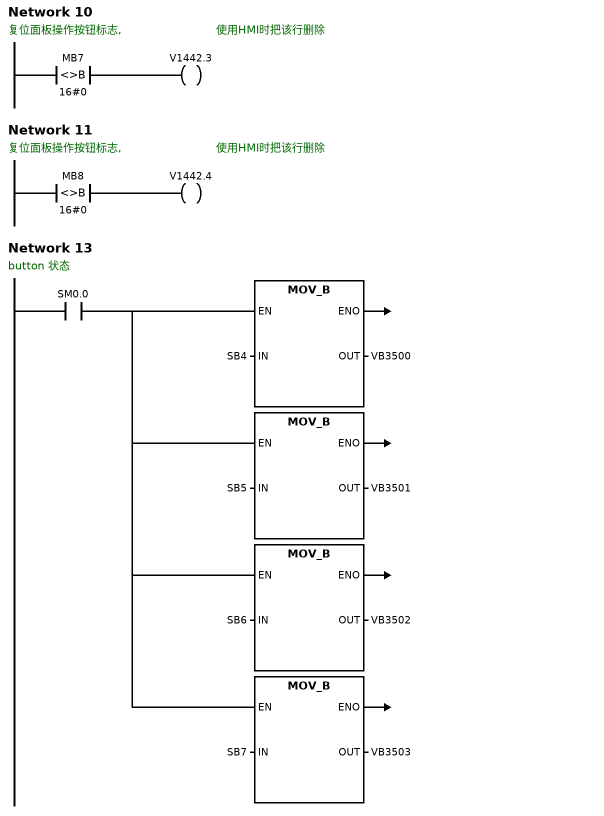
[picture p72: SBR17 networks 10-13]
Network 10
// 复位面板操作按钮标志,                           使用HMI时把该行删除
LDB<>  MB7, 16#0
=      V1442.3
Network 11
// 复位面板操作按钮标志,                           使用HMI时把该行删除
LDB<>  MB8, 16#0
=      V1442.4
Network 13
// button 状态
LD     SM0.0
MOVB   SB4, VB3500
MOVB   SB5, VB3501
MOVB   SB6, VB3502
MOVB   SB7, VB3503
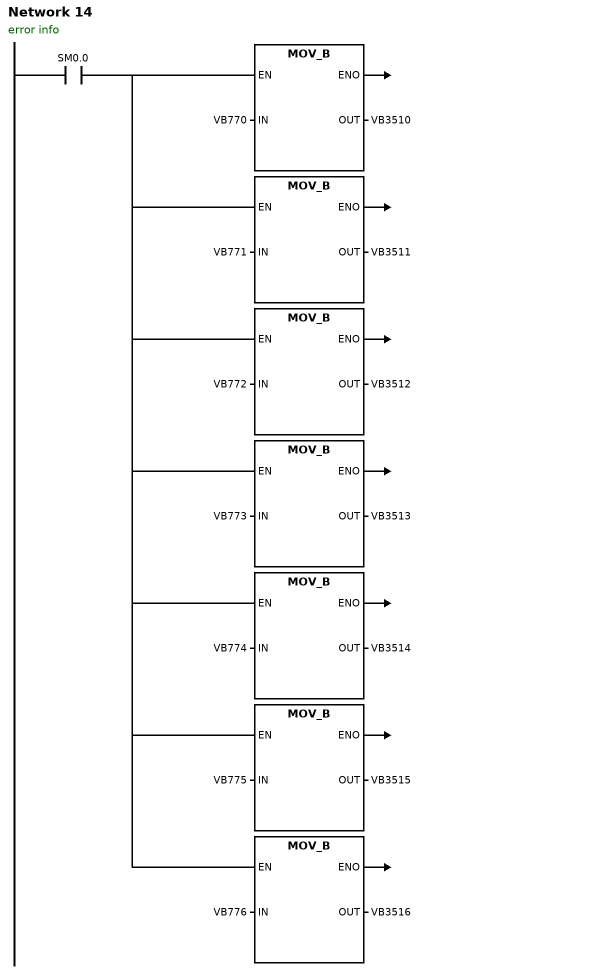
Network 14
// error info
LD     SM0.0
MOVB   VB770, VB3510
MOVB   VB771, VB3511
MOVB   VB772, VB3512
MOVB   VB773, VB3513
MOVB   VB774, VB3514
MOVB   VB775, VB3515
MOVB   VB776, VB3516
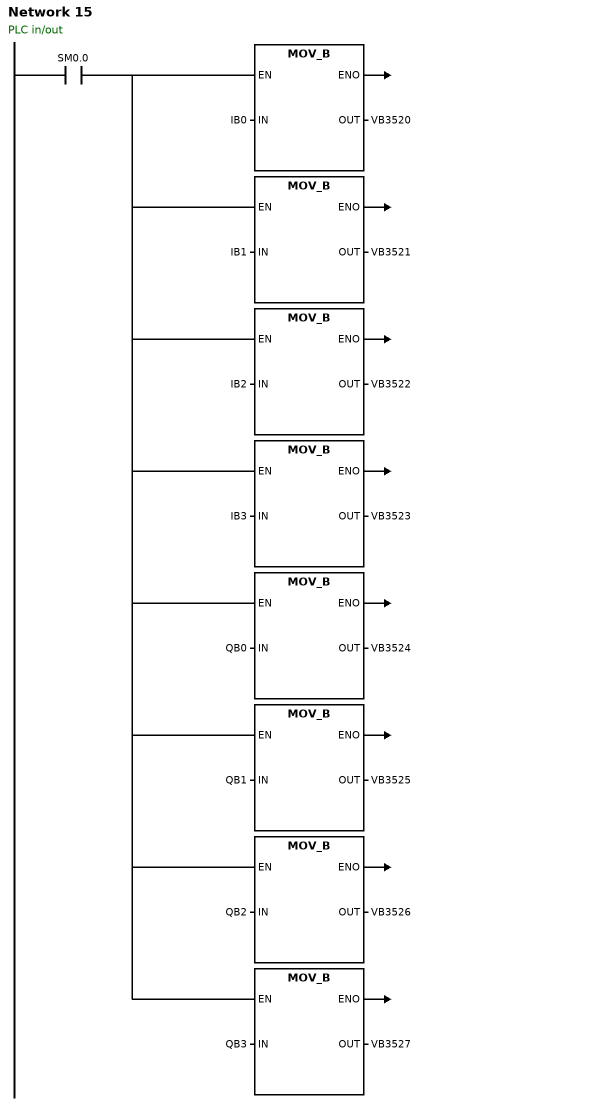
Network 15
// PLC in/out
LD     SM0.0
MOVB   IB0, VB3520
MOVB   IB1, VB3521
MOVB   IB2, VB3522
MOVB   IB3, VB3523
MOVB   QB0, VB3524
MOVB   QB1, VB3525
MOVB   QB2, VB3526
MOVB   QB3, VB3527
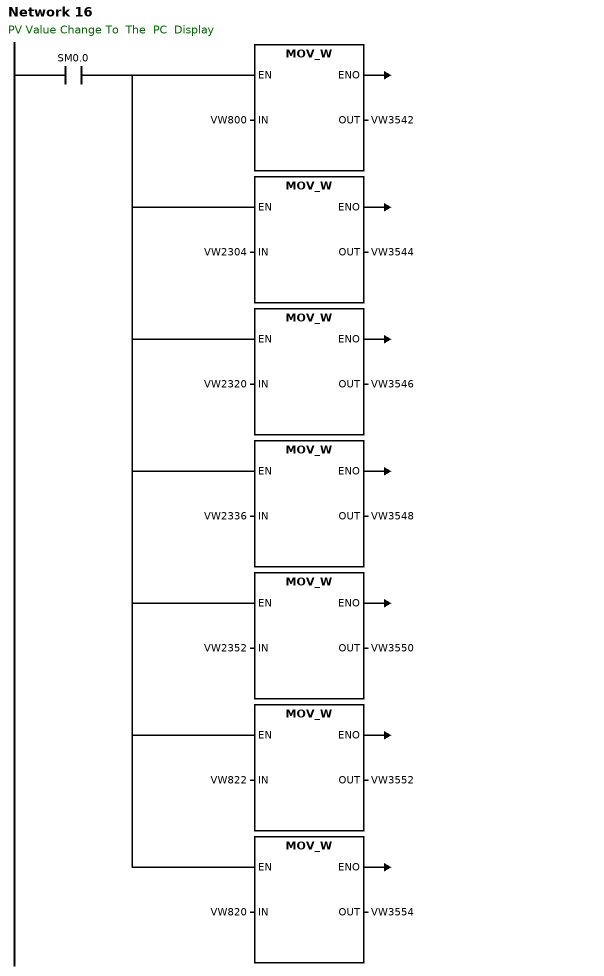
Network 16
// PV Value Change To  The  PC  Display 
LD     SM0.0
MOVW   VW800, VW3542
MOVW   VW2304, VW3544
MOVW   VW2320, VW3546
MOVW   VW2336, VW3548
MOVW   VW2352, VW3550
MOVW   VW822, VW3552
MOVW   VW820, VW3554
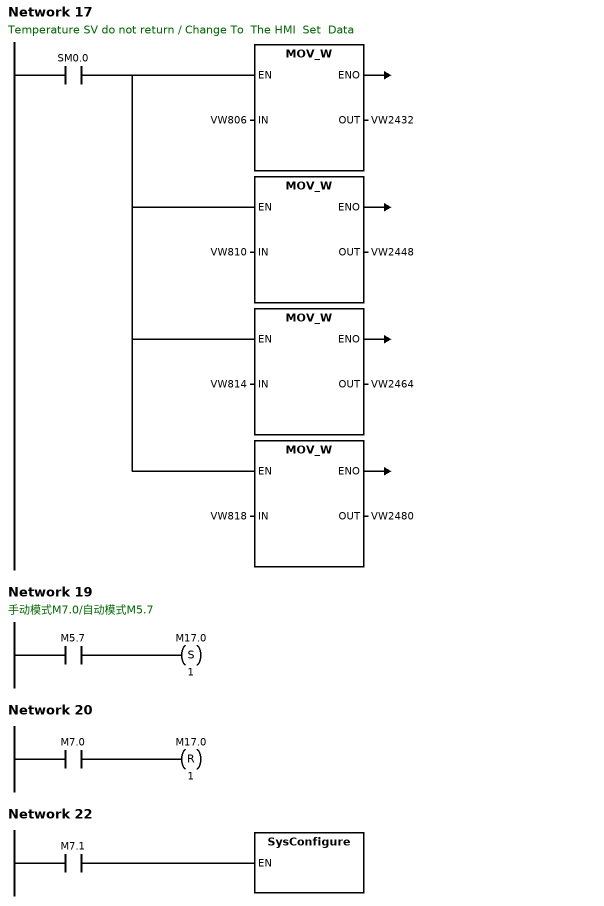
Network 17
// Temperature SV do not return
// Change To  The HMI  Set  Data  
LD     SM0.0
MOVW   VW806, VW2432
MOVW   VW810, VW2448
MOVW   VW814, VW2464
MOVW   VW818, VW2480
Network 18
// HMI PV Display
Network 19
// 手动模式M7.0/自动模式M5.7
LD     M5.7
S      M17.0, 1
Network 20
LD     M7.0
R      M17.0, 1
Network 21
// MB15     自动启动激活/失效在画面点OK是或后下载
Network 22
LD     M7.1
CALL   SysConfigure:SBR29
END_SUBROUTINE_BLOCK

SUBROUTINE_BLOCK DefaultValue:SBR18
TITLE=
BEGIN
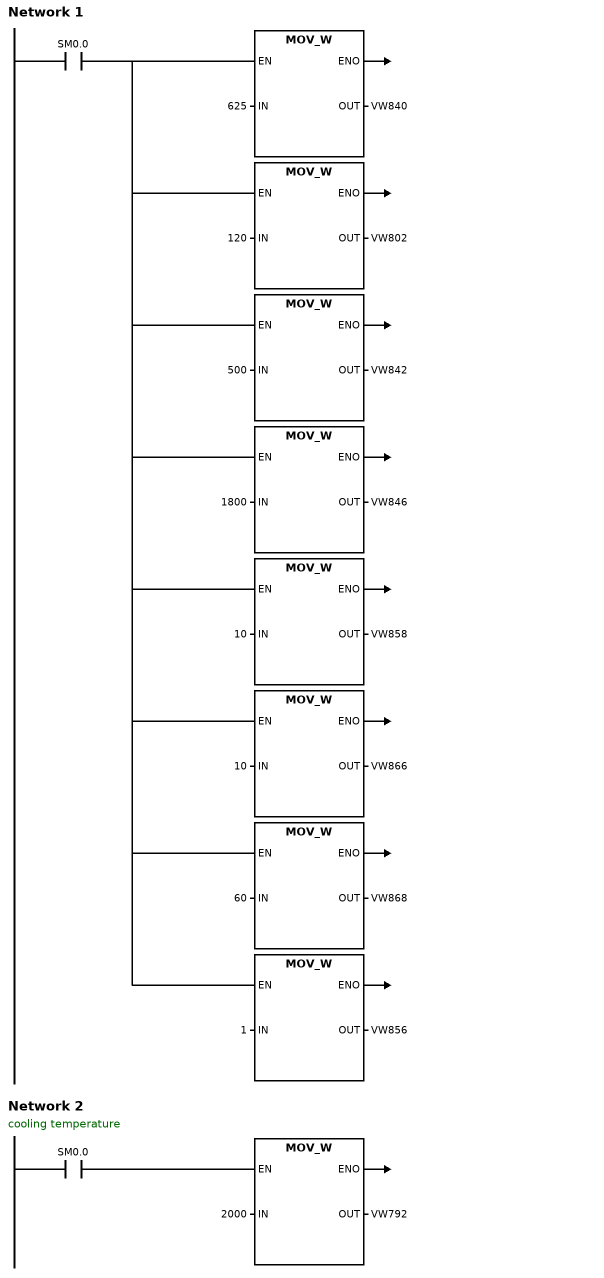
Network 1
LD     SM0.0
MOVW   625, VW840
MOVW   120, VW802
MOVW   500, VW842
MOVW   1800, VW846
MOVW   10, VW858
MOVW   10, VW866
MOVW   60, VW868
MOVW   1, VW856
Network 2
// cooling temperature
LD     SM0.0
MOVW   2000, VW792
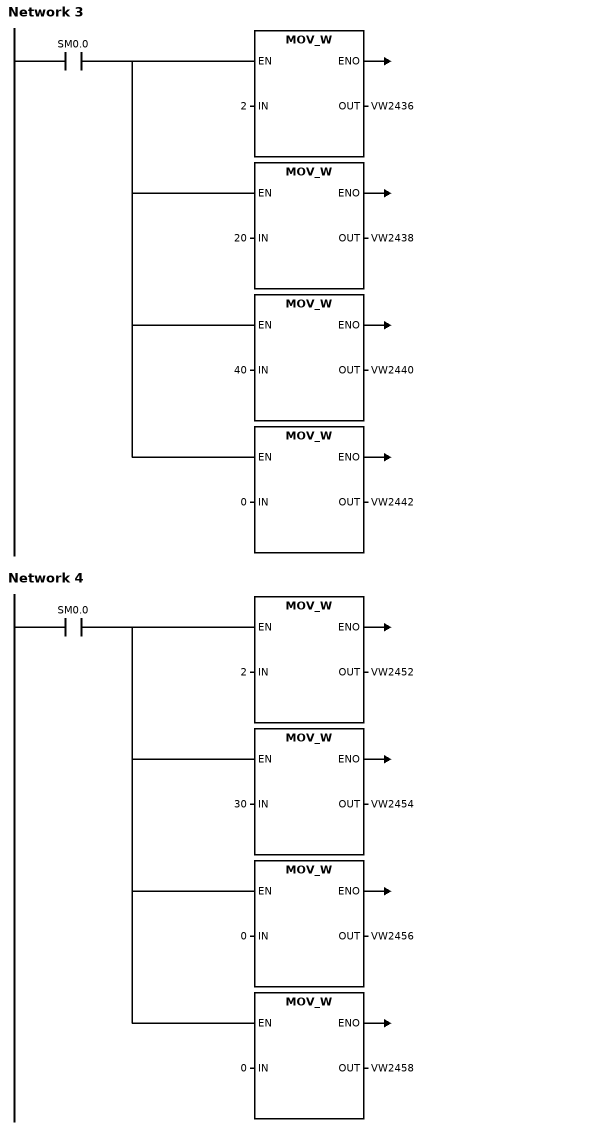
Network 3
LD     SM0.0
MOVW   2, VW2436
MOVW   20, VW2438
MOVW   40, VW2440
MOVW   0, VW2442
Network 4
LD     SM0.0
MOVW   2, VW2452
MOVW   30, VW2454
MOVW   0, VW2456
MOVW   0, VW2458
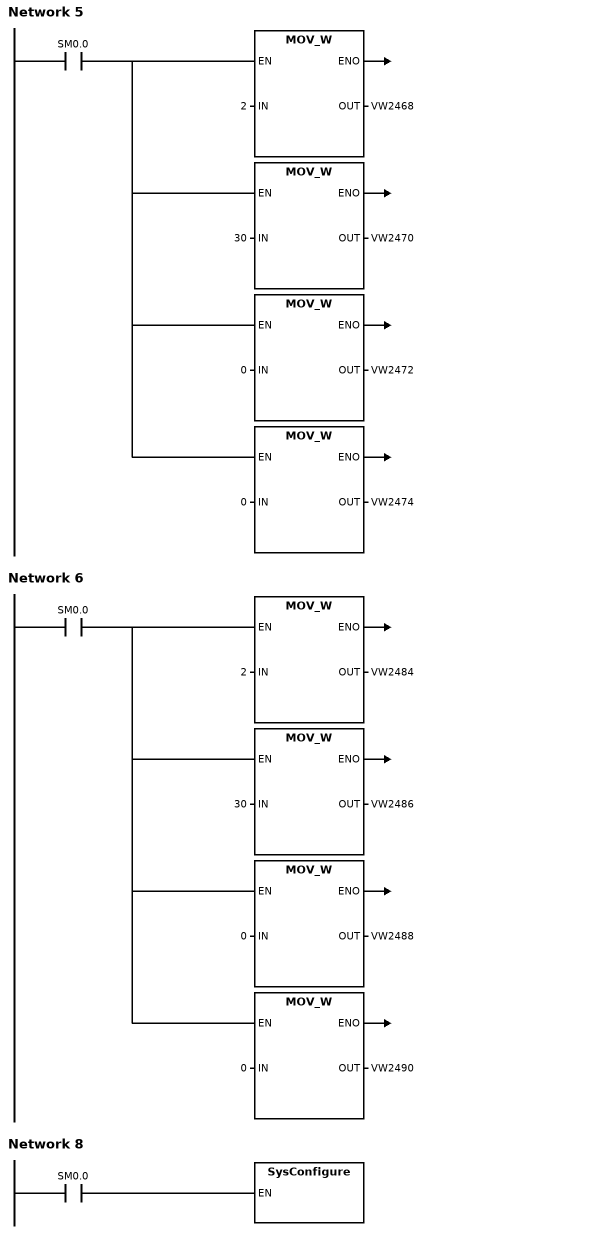
Network 5
LD     SM0.0
MOVW   2, VW2468
MOVW   30, VW2470
MOVW   0, VW2472
MOVW   0, VW2474
Network 6
LD     SM0.0
MOVW   2, VW2484
MOVW   30, VW2486
MOVW   0, VW2488
MOVW   0, VW2490
Network 8
LD     SM0.0
CALL   SysConfigure:SBR29
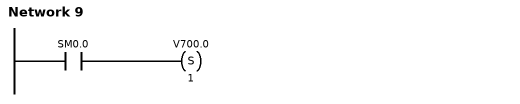
Network 9
LD     SM0.0
S      V700.0, 1
END_SUBROUTINE_BLOCK

SUBROUTINE_BLOCK ShiftingVB1000_1138:SBR19
TITLE=
BEGIN
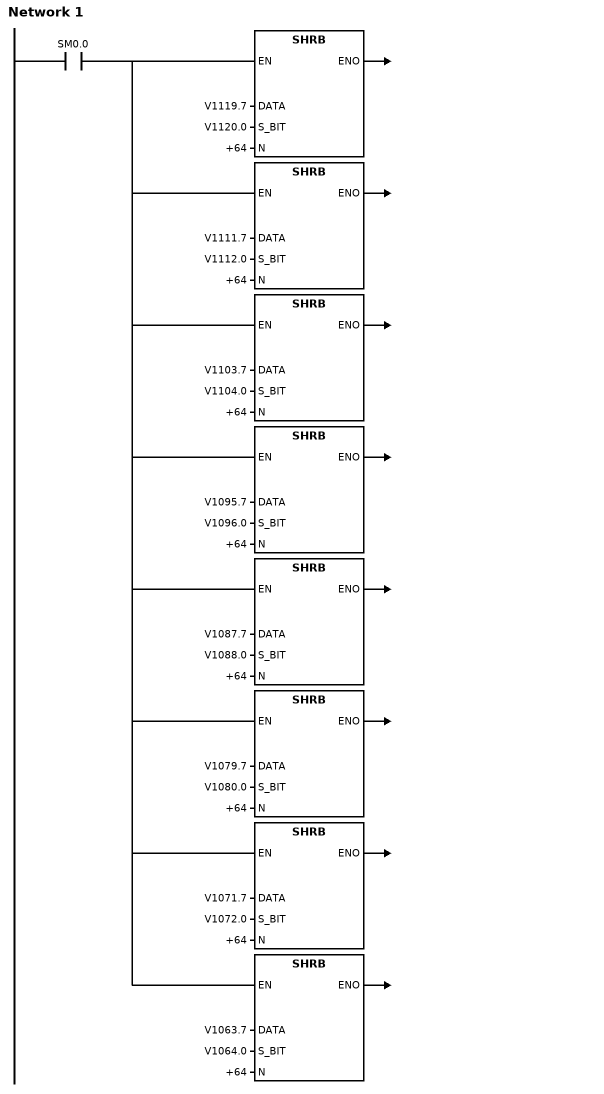
Network 1
LD     SM0.0
SHRB   V1119.7, V1120.0, +64
SHRB   V1111.7, V1112.0, +64
SHRB   V1103.7, V1104.0, +64
SHRB   V1095.7, V1096.0, +64
SHRB   V1087.7, V1088.0, +64
SHRB   V1079.7, V1080.0, +64
SHRB   V1071.7, V1072.0, +64
SHRB   V1063.7, V1064.0, +64
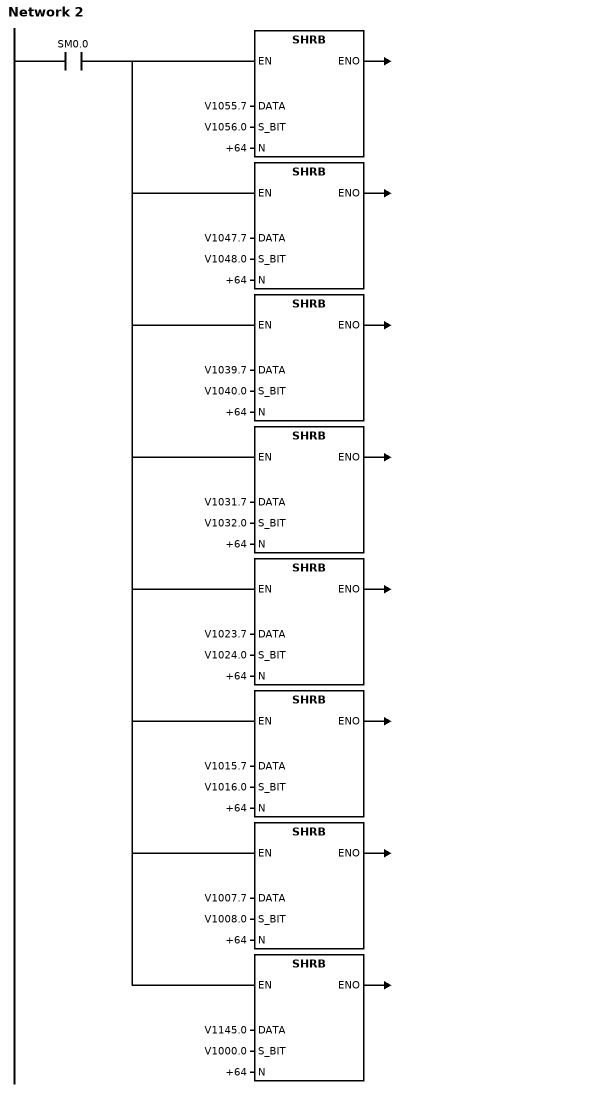
Network 2
LD     SM0.0
SHRB   V1055.7, V1056.0, +64
SHRB   V1047.7, V1048.0, +64
SHRB   V1039.7, V1040.0, +64
SHRB   V1031.7, V1032.0, +64
SHRB   V1023.7, V1024.0, +64
SHRB   V1015.7, V1016.0, +64
SHRB   V1007.7, V1008.0, +64
SHRB   V1145.0, V1000.0, +64
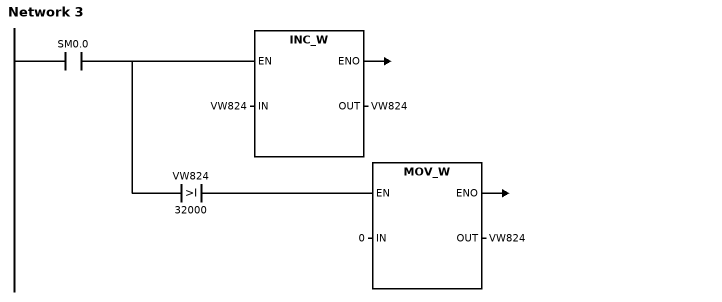
Network 3
LD     SM0.0
INCW   VW824
AW>    VW824, 32000
MOVW   0, VW824
END_SUBROUTINE_BLOCK

SUBROUTINE_BLOCK ConveySpeedInverter:SBR20
TITLE=
BEGIN
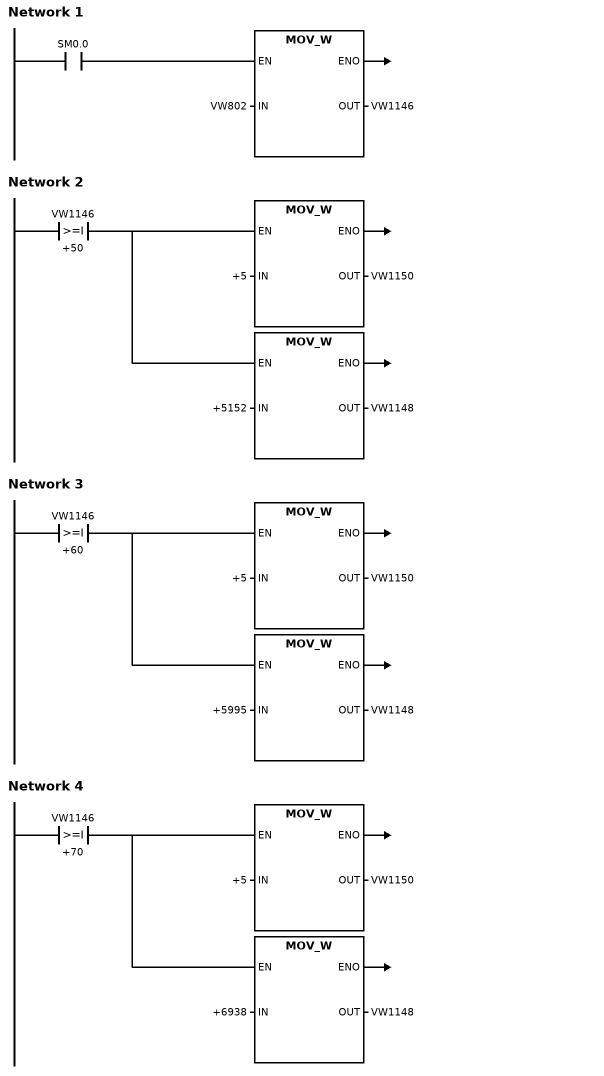
Network 1
LD     SM0.0
MOVW   VW802, VW1146
Network 2
LDW>=  VW1146, +50
MOVW   +5, VW1150
MOVW   +5152, VW1148
Network 3
LDW>=  VW1146, +60
MOVW   +5, VW1150
MOVW   +5995, VW1148
Network 4
LDW>=  VW1146, +70
MOVW   +5, VW1150
MOVW   +6938, VW1148
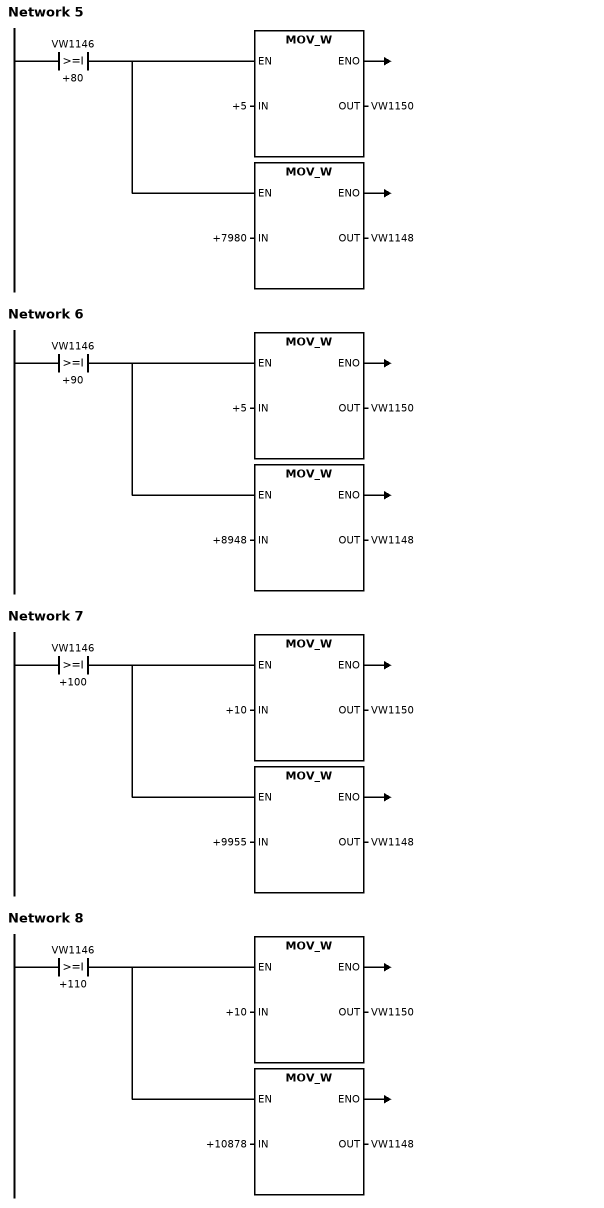
Network 5
LDW>=  VW1146, +80
MOVW   +5, VW1150
MOVW   +7980, VW1148
Network 6
LDW>=  VW1146, +90
MOVW   +5, VW1150
MOVW   +8948, VW1148
Network 7
LDW>=  VW1146, +100
MOVW   +10, VW1150
MOVW   +9955, VW1148
Network 8
LDW>=  VW1146, +110
MOVW   +10, VW1150
MOVW   +10878, VW1148
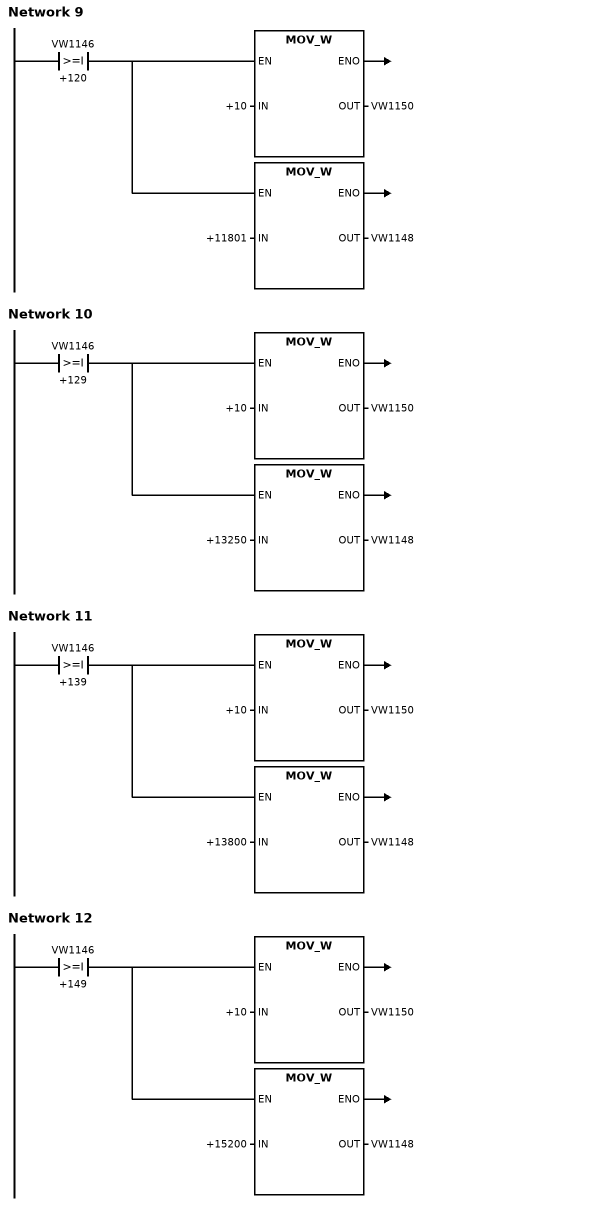
Network 9
LDW>=  VW1146, +120
MOVW   +10, VW1150
MOVW   +11801, VW1148
Network 10
LDW>=  VW1146, +129
MOVW   +10, VW1150
MOVW   +13250, VW1148
Network 11
LDW>=  VW1146, +139
MOVW   +10, VW1150
MOVW   +13800, VW1148
Network 12
LDW>=  VW1146, +149
MOVW   +10, VW1150
MOVW   +15200, VW1148
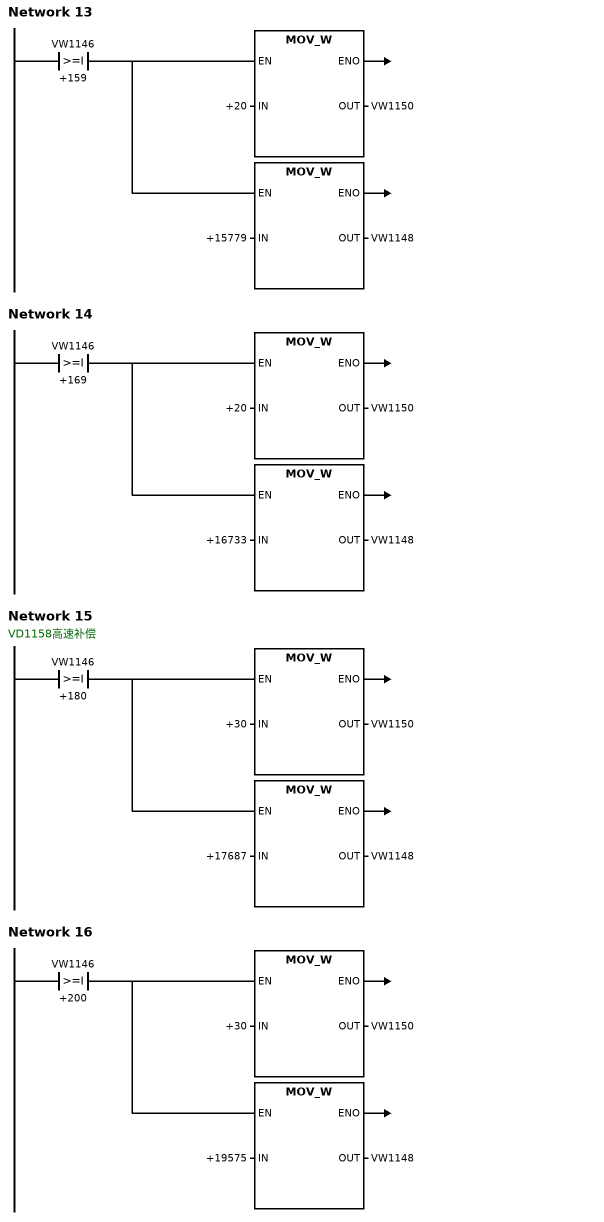
Network 13
LDW>=  VW1146, +159
MOVW   +20, VW1150
MOVW   +15779, VW1148
Network 14
LDW>=  VW1146, +169
MOVW   +20, VW1150
MOVW   +16733, VW1148
Network 15
// VD1158高速补偿
LDW>=  VW1146, +180
MOVW   +30, VW1150
MOVW   +17687, VW1148
Network 16
LDW>=  VW1146, +200
MOVW   +30, VW1150
MOVW   +19575, VW1148
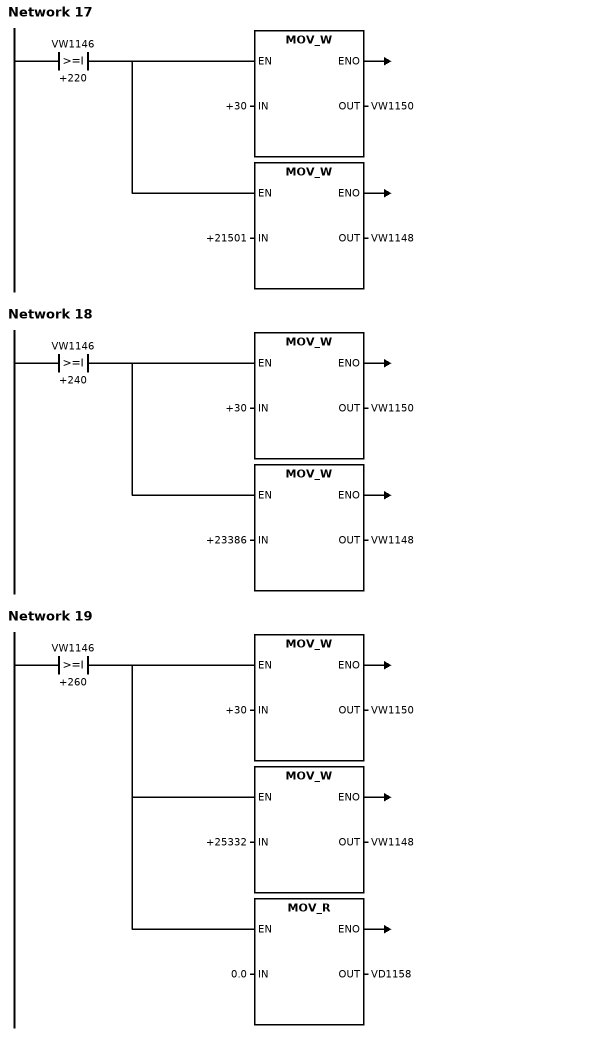
Network 17
LDW>=  VW1146, +220
MOVW   +30, VW1150
MOVW   +21501, VW1148
Network 18
LDW>=  VW1146, +240
MOVW   +30, VW1150
MOVW   +23386, VW1148
Network 19
LDW>=  VW1146, +260
MOVW   +30, VW1150
MOVW   +25332, VW1148
MOVR   0.0, VD1158
END_SUBROUTINE_BLOCK

SUBROUTINE_BLOCK ConveySpeedDV1234:SBR21
TITLE=
BEGIN
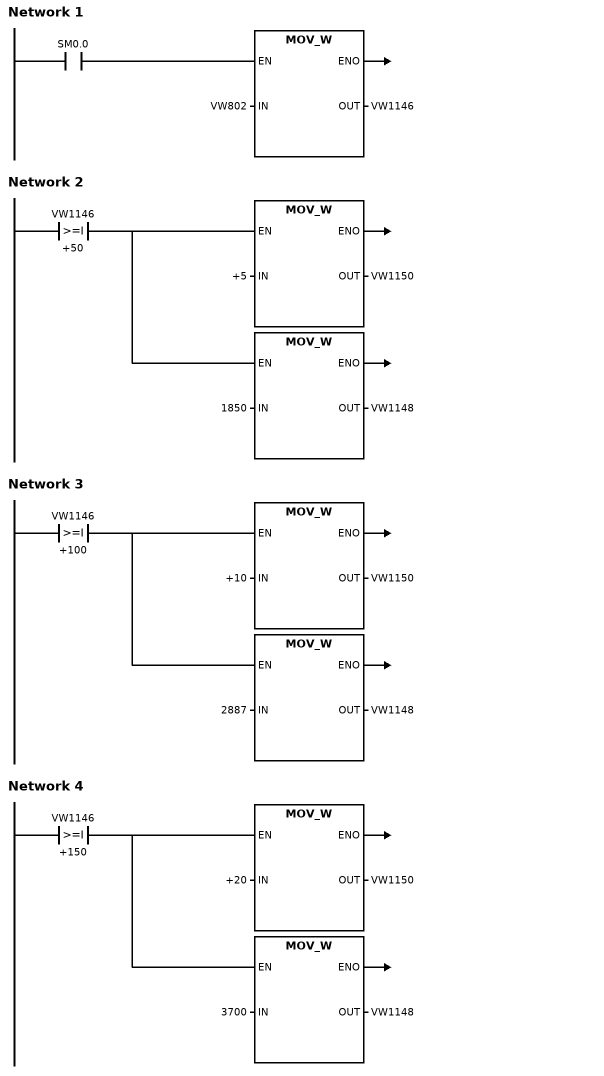
Network 1
LD     SM0.0
MOVW   VW802, VW1146
Network 2
LDW>=  VW1146, +50
MOVW   +5, VW1150
MOVW   1850, VW1148
Network 3
LDW>=  VW1146, +100
MOVW   +10, VW1150
MOVW   2887, VW1148
Network 4
LDW>=  VW1146, +150
MOVW   +20, VW1150
MOVW   3700, VW1148
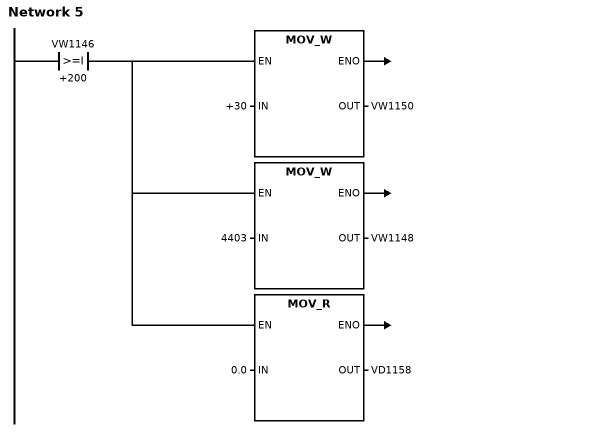
Network 5
LDW>=  VW1146, +200
MOVW   +30, VW1150
MOVW   4403, VW1148
MOVR   0.0, VD1158
END_SUBROUTINE_BLOCK

SUBROUTINE_BLOCK WagChangeSpeed:SBR22
TITLE=
BEGIN
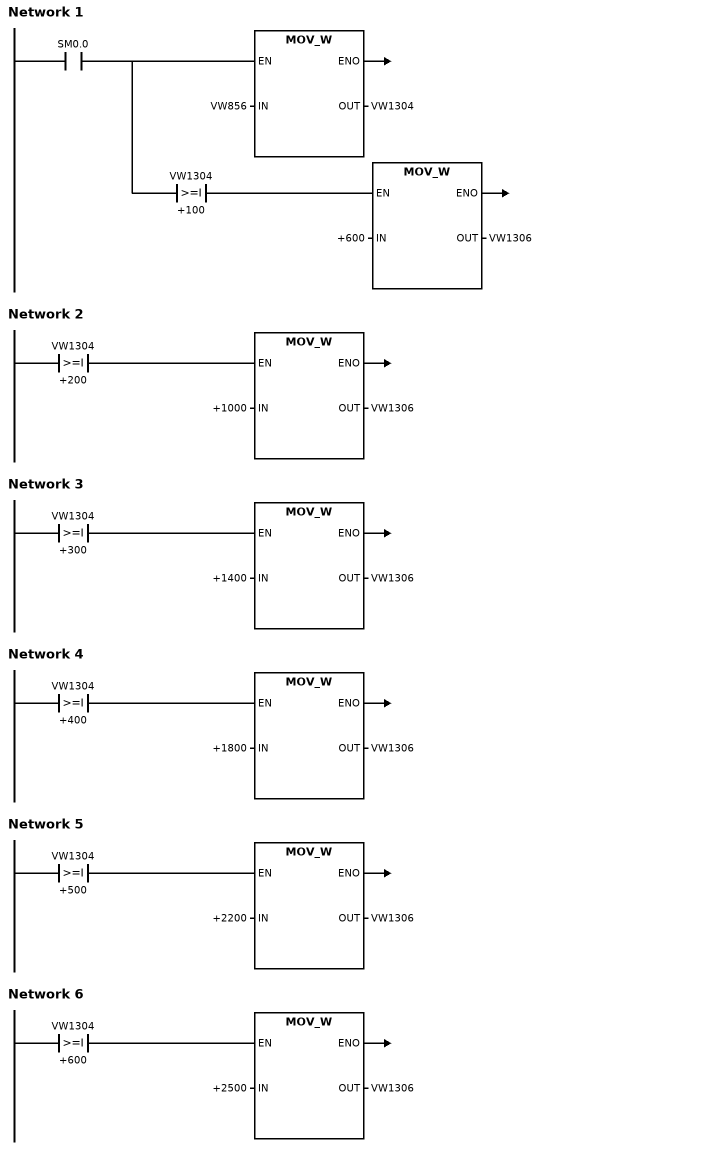
Network 1
LD     SM0.0
MOVW   VW856, VW1304
AW>=   VW1304, +100
MOVW   +600, VW1306
Network 2
LDW>=  VW1304, +200
MOVW   +1000, VW1306
Network 3
LDW>=  VW1304, +300
MOVW   +1400, VW1306
Network 4
LDW>=  VW1304, +400
MOVW   +1800, VW1306
Network 5
LDW>=  VW1304, +500
MOVW   +2200, VW1306
Network 6
LDW>=  VW1304, +600
MOVW   +2500, VW1306
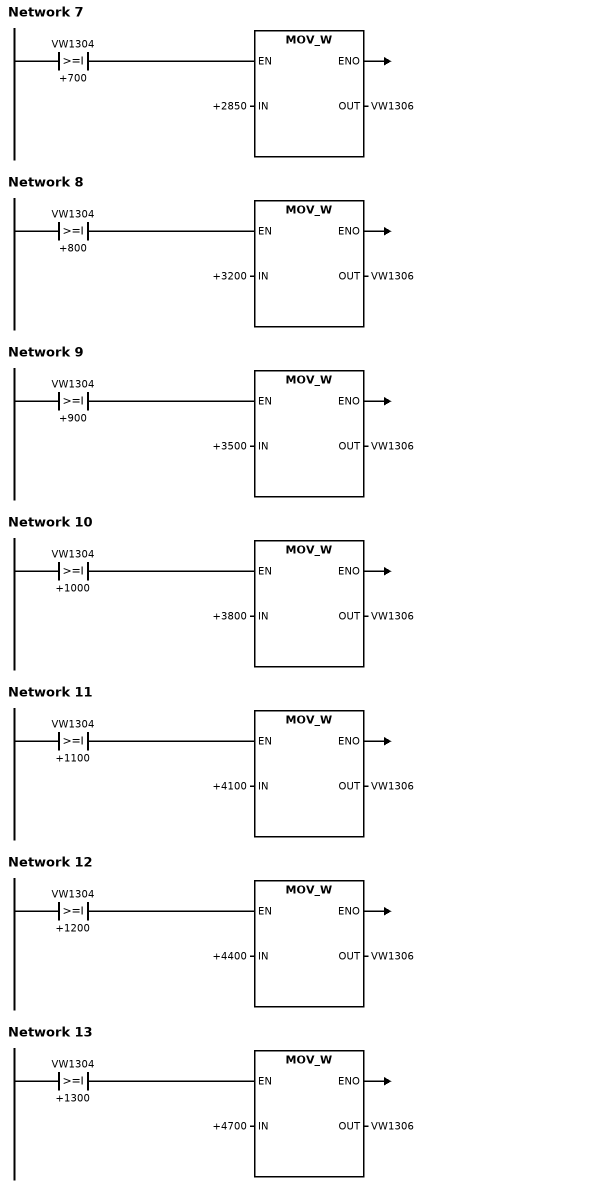
Network 7
LDW>=  VW1304, +700
MOVW   +2850, VW1306
Network 8
LDW>=  VW1304, +800
MOVW   +3200, VW1306
Network 9
LDW>=  VW1304, +900
MOVW   +3500, VW1306
Network 10
LDW>=  VW1304, +1000
MOVW   +3800, VW1306
Network 11
LDW>=  VW1304, +1100
MOVW   +4100, VW1306
Network 12
LDW>=  VW1304, +1200
MOVW   +4400, VW1306
Network 13
LDW>=  VW1304, +1300
MOVW   +4700, VW1306
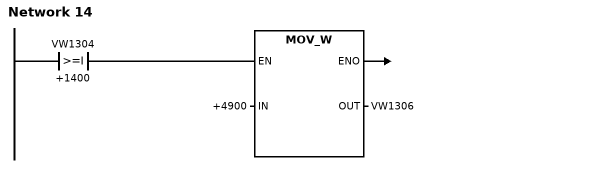
Network 14
LDW>=  VW1304, +1400
MOVW   +4900, VW1306
END_SUBROUTINE_BLOCK

SUBROUTINE_BLOCK WaveChangeSpeed:SBR23
TITLE=
BEGIN
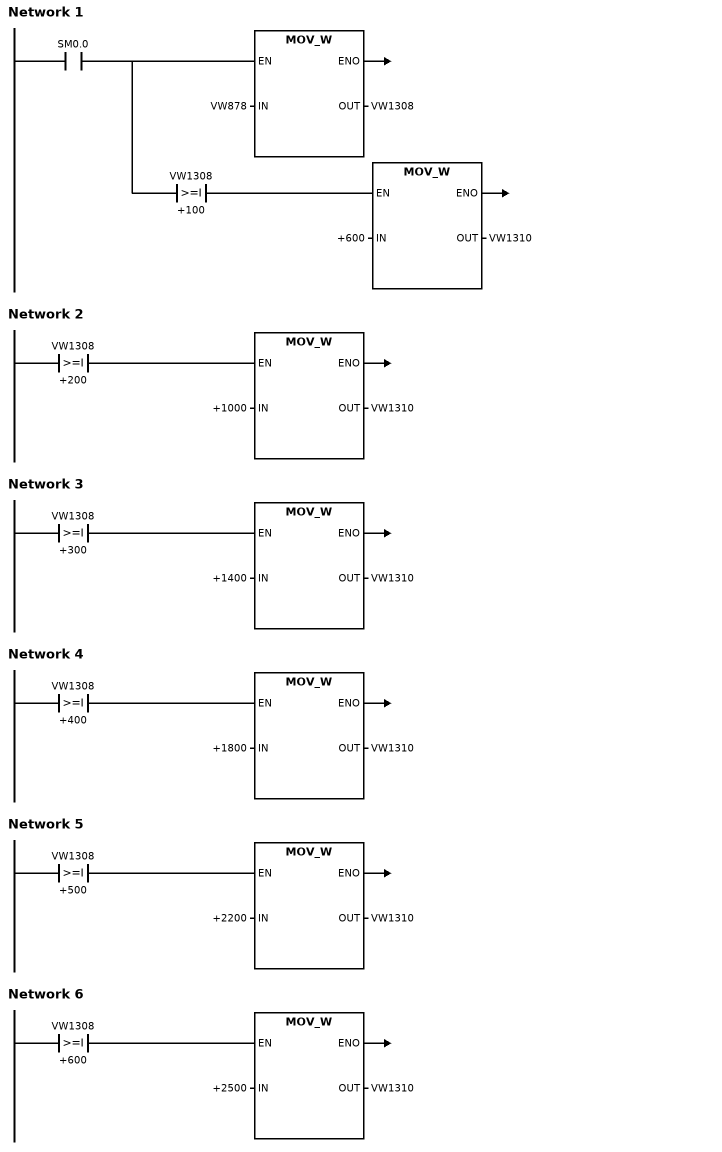
Network 1
LD     SM0.0
MOVW   VW878, VW1308
AW>=   VW1308, +100
MOVW   +600, VW1310
Network 2
LDW>=  VW1308, +200
MOVW   +1000, VW1310
Network 3
LDW>=  VW1308, +300
MOVW   +1400, VW1310
Network 4
LDW>=  VW1308, +400
MOVW   +1800, VW1310
Network 5
LDW>=  VW1308, +500
MOVW   +2200, VW1310
Network 6
LDW>=  VW1308, +600
MOVW   +2500, VW1310
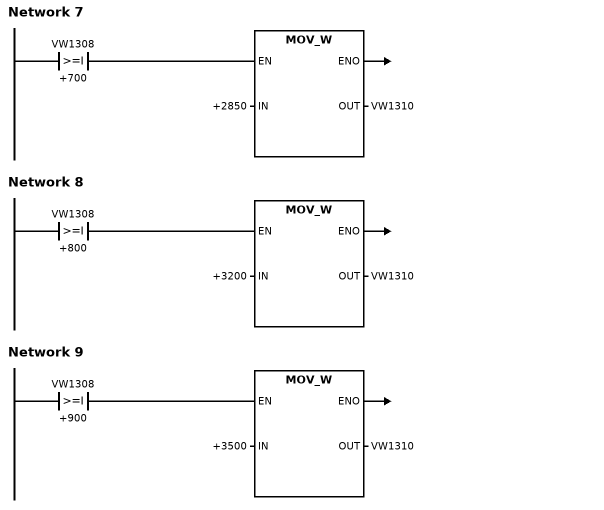
Network 7
LDW>=  VW1308, +700
MOVW   +2850, VW1310
Network 8
LDW>=  VW1308, +800
MOVW   +3200, VW1310
Network 9
LDW>=  VW1308, +900
MOVW   +3500, VW1310
END_SUBROUTINE_BLOCK

SUBROUTINE_BLOCK SpewChangeSpeed:SBR24
TITLE=
BEGIN
